PROGRAM GL7_Conveyor
VAR
	
	RUN_FWD_BIT_TO_EXIT : BOOL; // RUN FORWARD TO EXIT POSITION AFTER DROP
END_VAR
VAR // added by the converter: edge detectors and wires of the graphical bodies
    _w1 : BOOL;
END_VAR

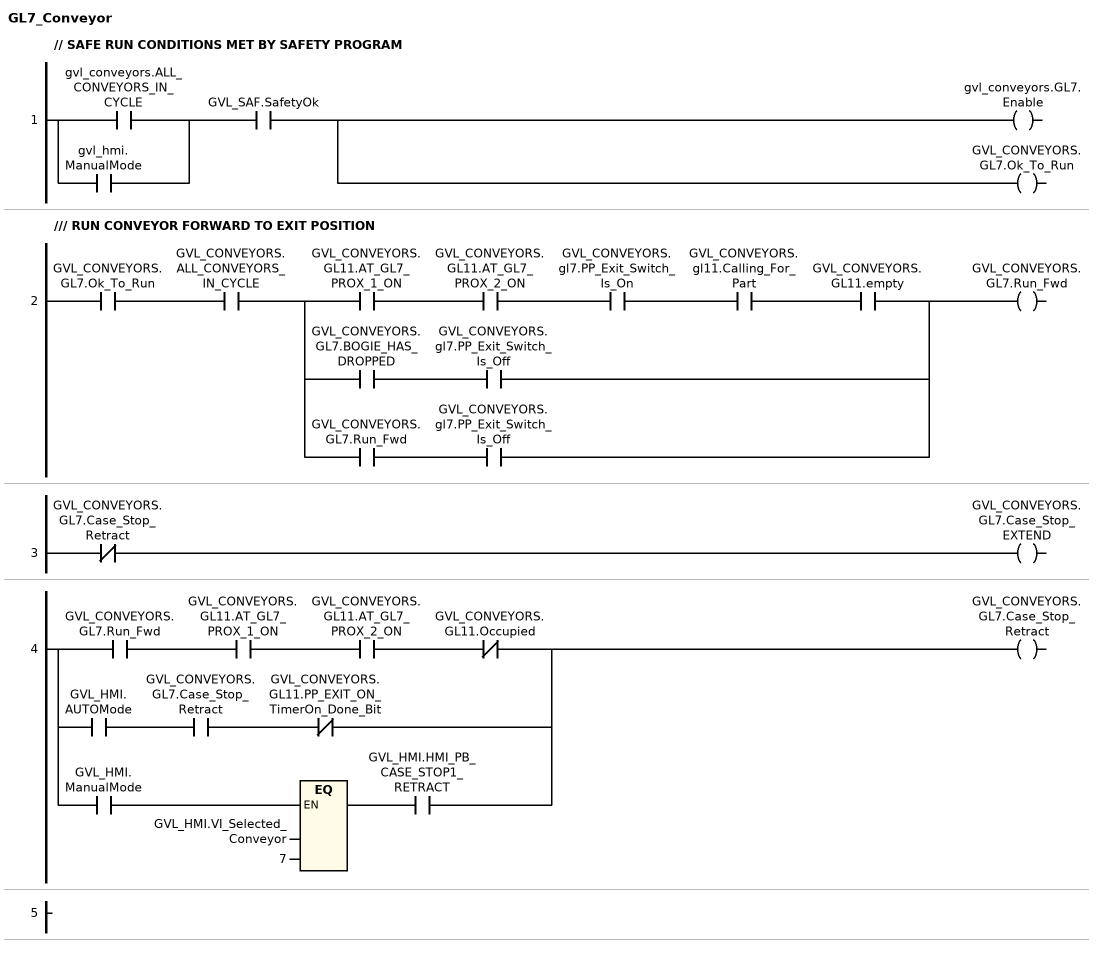
// NETWORK 1: // SAFE RUN CONDITIONS MET BY SAFETY PROGRAM
_w1 := (gvl_conveyors.ALL_CONVEYORS_IN_CYCLE OR gvl_hmi.ManualMode) AND GVL_SAF.SafetyOk;
gvl_conveyors.GL7.Enable := _w1;
GVL_CONVEYORS.GL7.Ok_To_Run := _w1;

// NETWORK 2: /// RUN CONVEYOR FORWARD TO EXIT POSITION
GVL_CONVEYORS.GL7.Run_Fwd := GVL_CONVEYORS.GL7.Ok_To_Run AND GVL_CONVEYORS.ALL_CONVEYORS_IN_CYCLE AND (GVL_CONVEYORS.GL11.AT_GL7_PROX_1_ON AND GVL_CONVEYORS.GL11.AT_GL7_PROX_2_ON AND GVL_CONVEYORS.gl7.PP_Exit_Switch_Is_On AND GVL_CONVEYORS.gl11.Calling_For_Part AND GVL_CONVEYORS.GL11.empty OR GVL_CONVEYORS.GL7.BOGIE_HAS_DROPPED AND GVL_CONVEYORS.gl7.PP_Exit_Switch_Is_Off OR GVL_CONVEYORS.GL7.Run_Fwd AND GVL_CONVEYORS.gl7.PP_Exit_Switch_Is_Off);

// NETWORK 3
GVL_CONVEYORS.GL7.Case_Stop_EXTEND := NOT GVL_CONVEYORS.GL7.Case_Stop_Retract;

// NETWORK 4
GVL_CONVEYORS.GL7.Case_Stop_Retract := GVL_CONVEYORS.GL7.Run_Fwd AND GVL_CONVEYORS.GL11.AT_GL7_PROX_1_ON AND GVL_CONVEYORS.GL11.AT_GL7_PROX_2_ON AND NOT GVL_CONVEYORS.GL11.Occupied OR GVL_HMI.AUTOMode AND GVL_CONVEYORS.GL7.Case_Stop_Retract AND NOT GVL_CONVEYORS.GL11.PP_EXIT_ON_TimerOn_Done_Bit OR (GVL_HMI.ManualMode AND GVL_HMI.VI_Selected_Conveyor = 7) AND GVL_HMI.HMI_PB_CASE_STOP1_RETRACT;

// NETWORK 5

END_PROGRAM

(* stored: Version 1.1.0.1, ProductVersion 3.1.4024.12
   POU GL7_Conveyor: Id {3c1ba7ad-bd9c-41b5-ad8a-cf216df4f818}, SpecialFunc None *)
